// TwinCAT 3 PLC project Prototype_version2
// ProgramVersion: 3.1.4024.0
// libraries:
//   Tc2_Standard, * (Beckhoff Automation GmbH)
//   Tc2_System, * (Beckhoff Automation GmbH)
//   Tc3_Module, * (Beckhoff Automation GmbH)
// project tree:
//   / Class Diagram.TcCD (not stored), PlcTask.TcTTO
//   Classes/ Circle.TcPOU, Disposable.TcPOU, Rectangle.TcPOU
//   Interfaces/ I_Disposable.TcIO, I_DrawableShape.TcIO
//   POUs/ MAIN.TcPOU
// real-time tasks:
//   TASK PlcTask: cycle T#10ms, priority 20, ADS port 350

CONFIGURATION Prototype_version2
    RESOURCE PLC ON TwinCAT3
        TASK PlcTask(INTERVAL := T#10ms, PRIORITY := 20);
        PROGRAM MAIN WITH PlcTask : MAIN;
    END_RESOURCE
END_CONFIGURATION

// ---- Interfaces/I_Disposable.TcIO
INTERFACE I_Disposable

METHOD Dispose
VAR_INPUT
END_VAR
END_METHOD

END_INTERFACE

// ---- Interfaces/I_DrawableShape.TcIO
INTERFACE I_DrawableShape EXTENDS I_Disposable

METHOD Clone : I_DrawableShape
VAR_INPUT
END_VAR
END_METHOD

METHOD Draw
VAR_INPUT
END_VAR
END_METHOD

END_INTERFACE

// ---- POUs/MAIN.TcPOU
PROGRAM MAIN
VAR
    originalRectangle: Rectangle;
    clonedRectangle: I_DrawableShape;
	
    originalCircle: Circle;
    clonedCircle: I_DrawableShape;
	
	bRequest : BOOL;
	counter: INT;

END_VAR

// https://refactoring.guru/design-patterns/prototype

// Recuerda que el patrón Prototipo permite crear nuevos objetos clonando un objeto existente, evitando así la necesidad de crear nuevas instancias desde cero.

// porque salen varios mensajes:
// https://github.com/tcunit/TcUnit/issues/92
// solución temporal : Unload project...
IF bRequest THEN
	
	// rectangle example 
	originalRectangle.width := 10;
	originalRectangle.height := 5;
	originalRectangle.Draw();
	clonedRectangle := originalRectangle.clone();
	clonedRectangle.Draw();
	clonedRectangle.Dispose(); 
	
	// circle example 
	originalCircle.radius := 7;
	originalCircle.Draw();
	clonedCircle := originalCircle.clone();
	clonedCircle.Draw();
	clonedCircle.Dispose(); 
	
	// report request info
	bRequest := FALSE;
	counter := counter + 1;
	ADSLOGSTR(msgCtrlMask :=ADSLOG_MSGTYPE_HINT, msgFmtStr :='test: %s', strArg := TO_STRING(counter));

END_IF

END_PROGRAM

// ---- Classes/Rectangle.TcPOU
{attribute 'enable_dynamic_creation'}
FUNCTION_BLOCK Rectangle EXTENDS Disposable IMPLEMENTS I_DrawableShape
VAR
	_width: INT;
    _height: INT;
END_VAR

METHOD Clone : I_DrawableShape
VAR
	pRectangle : POINTER TO Rectangle;
END_VAR
pRectangle := __NEW(Rectangle);
pRectangle^.Width := Width;
pRectangle^.Height := Height;
Clone := pRectangle^;
END_METHOD

METHOD Draw
VAR
	str_width : STRING;
	str_height : STRING;
	str : STRING;
END_VAR
str_width := CONCAT(STR1 := 'width: ', STR2 := TO_STRING(Width));
str_height := CONCAT(STR1 := 'height: ', STR2 := TO_STRING(Height));
str := CONCAT(STR1 := str_width, STR2 := str_height);
ADSLOGSTR(msgCtrlMask := ADSLOG_MSGTYPE_HINT, msgFmtStr := 'Draw Rectangle with:  %s', strArg := str);
END_METHOD

PROPERTY PUBLIC Height : INT
GET
Height := _height;
END_GET
SET // PUBLIC
_height := Height;
END_SET
END_PROPERTY

PROPERTY PUBLIC Width : INT
GET
Width := _width;
END_GET
SET // PUBLIC
_width := Width;
END_SET
END_PROPERTY

END_FUNCTION_BLOCK

// ---- Classes/Disposable.TcPOU
FUNCTION_BLOCK Disposable
VAR
END_VAR

METHOD PUBLIC Dispose
VAR_INPUT
END_VAR
__DELETE(THIS);
END_METHOD

END_FUNCTION_BLOCK

// ---- Classes/Circle.TcPOU
{attribute 'enable_dynamic_creation'}
FUNCTION_BLOCK Circle EXTENDS Disposable IMPLEMENTS I_DrawableShape
VAR
	_radius: INT;
END_VAR

METHOD Clone : I_DrawableShape
VAR
	pCircle : POINTER TO Circle;	
END_VAR
pCircle := __NEW(Circle);
pCircle^.radius := radius;
Clone := pCircle^;
END_METHOD


METHOD Draw

VAR
	str : STRING;
END_VAR
str := TO_STRING(radius);
ADSLOGSTR(msgCtrlMask :=ADSLOG_MSGTYPE_HINT, msgFmtStr :='Draw circle with radius: %s', strArg := str);
END_METHOD

PROPERTY Radius : INT
GET
Radius := _radius;
END_GET
SET
_radius := Radius;
END_SET
END_PROPERTY

END_FUNCTION_BLOCK
